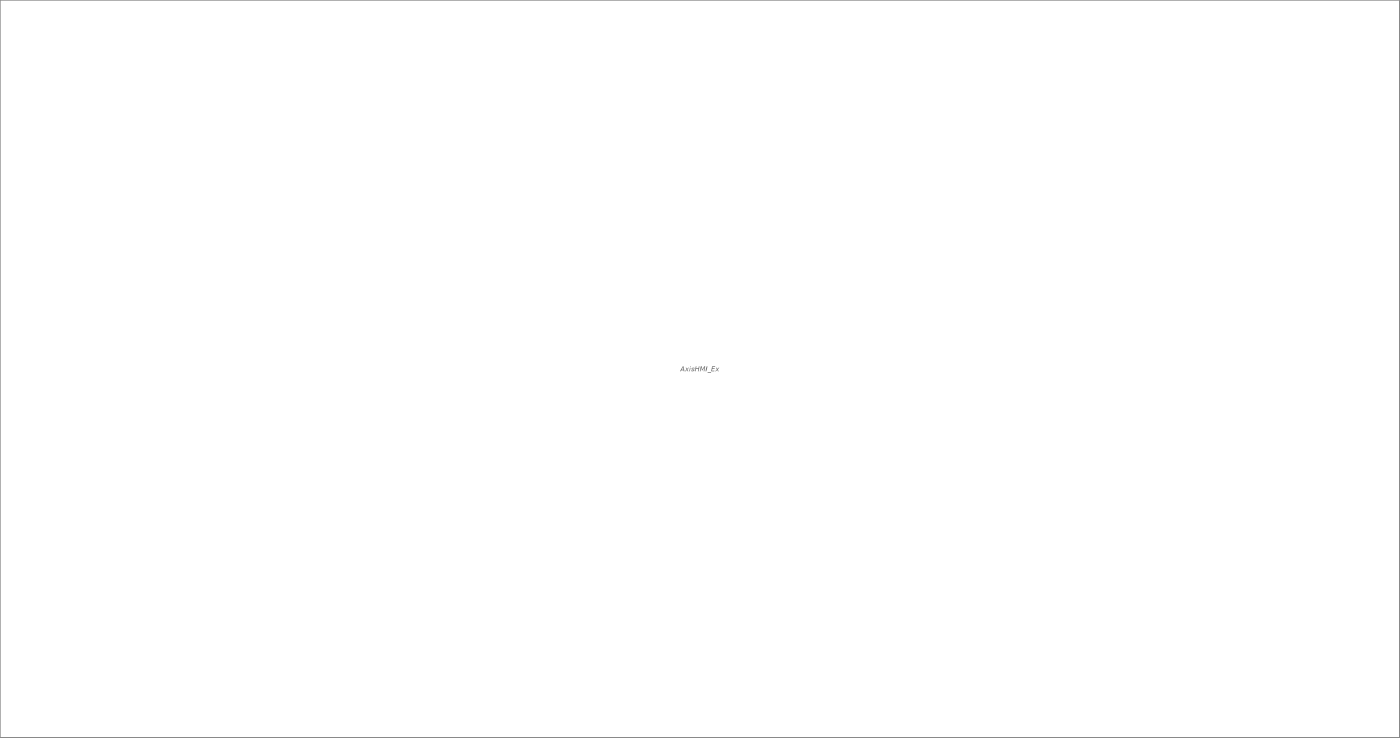
VISUALIZATION visu_buffer  // 2048x1080
    TabControl (0,0 2048x1080)
        shows AxisHMI_Ex(stAxisHMI := GVL.fb_buffer.fb_rollers[3].st_mcAxis, mcAxis := GVL.fb_buffer.fb_rollers[3].mcAxis, xError := GVL.fb_buffer.fb_rollers[3].mcAxis.xError)
        shows v_io_buffer()
        shows Axis_HMI(st_axis_HMI := st_mcAxis[EN_Axis.Grip_axis])
        shows AxisMotionLib.AxisHMI_Ex(stAxisHMI := gantrybase.st_mcAxis[EN_Axis.Z], mcAxis := gantrybase.mcAxis[EN_Axis.Z], xError := gantrybase.mcAxis[EN_Axis.Z].xError)
        shows v_rem_1(dIO_ReM := GVL.rem[G_HMI.iReM])
        [0]: TabTitle=Buffer Stopper
        [6]: TabTitle=Gripper
        [1]: AxisHMI=gantrybase.st_mcAxis[EN_Axis.Y], mcAxis=gantrybase.mcAxis[EN_Axis.Y], Error=gantrybase.mcAxis[EN_Axis.Y].xError
        [3]: TabTitle=ReMIO_1
        p699000190: gantrybase.st_mcAxis[EN_Axis.X]
        p2837713833: gantrybase.mcAxis[EN_Axis.Z].sAxisName
        p520277221: gantrybase.mcAxis[EN_Axis.X].xError
        p3331604638: gantrybase.st_mcAxis[EN_Axis.Z]
        p1813558639: gantrybase.mcAxis[EN_Axis.Z].xError
        p1563495665: gantrybase.st_mcAxis[EN_Axis.Y]
        p2070126892: gantrybase.mcAxis[EN_Axis.Y].xError
        p3435970784: gantrybase.mcAxis[EN_Axis.X]
        p2829954345: gantrybase.mcAxis[EN_Axis.Y]
        p3218520426: gantrybase.mcAxis[EN_Axis.Z]
END_VISUALIZATION

(* stored: Version 1.1.0.1, ProductVersion 3.1.4024.12
   Visu visu_buffer: Id {4a2c74dd-6e4c-4dbf-b80f-55c88e9652a0} *)
